// Mitsubishi GX Works2 project: Class4_Signal   PLC: Q03UD

PROGRAM MAIN
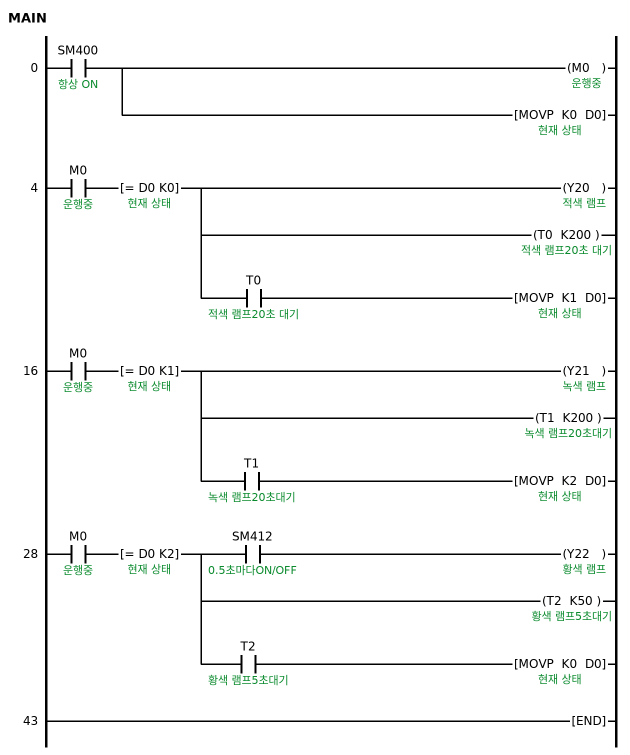
0     LD      SM400  ; 항상 ON
      OUT     M0  ; 운행중
      MOVP    K0 D0  ; 현재 상태
4     LD      M0  ; 운행중
      AND=    D0 K0  ; 현재 상태
      OUT     Y20  ; 적색 램프
      OUT     T0 K200  ; 적색 램프20초 대기
      AND     T0  ; 적색 램프20초 대기
      MOVP    K1 D0
16    LD      M0  ; 운행중
      AND=    D0 K1  ; 현재 상태
      OUT     Y21  ; 녹색 램프
      OUT     T1 K200  ; 녹색 램프20초대기
      AND     T1  ; 녹색 램프20초대기
      MOVP    K2 D0
28    LD      M0  ; 운행중
      AND=    D0 K2  ; 현재 상태
      MPS
      AND     SM412  ; 0.5초마다ON/OFF
      OUT     Y22  ; 황색 램프
      MPP
      OUT     T2 K50  ; 황색 램프5초대기
      AND     T2  ; 황색 램프5초대기
      MOVP    K0 D0
43    END
END_PROGRAM
